FUNCTION ASSEMBLE_LWORD_FROM_DWORDS (* this Function combines the 2 DWORDS to a LWORD *)
  (* Standard: 61499-1; Description: Copyright (c) 2026 HR Agrartechnik GmbH This program and the accompanying materials are made available under the terms of the Eclipse Public License 2.0 which is available at https://www.eclipse.org/legal/epl-2.0/ SPDX-License-Identifier: EPL-2.0 *)
  (* Version 1.0, 2026-05-16, Franz Höpfinger, HR Agrartechnik, initial Implementation *)
  PACKAGE eclipse4diac::utils::assembling;
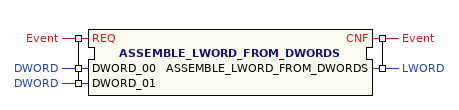
  EVENT_INPUT
    REQ WITH DWORD_00, DWORD_01;
  END_EVENT
  EVENT_OUTPUT
    CNF WITH ASSEMBLE_LWORD_FROM_DWORDS;
  END_EVENT
  VAR_INPUT
    DWORD_00 : DWORD;
    DWORD_01 : DWORD;
  END_VAR
  VAR_OUTPUT
    ASSEMBLE_LWORD_FROM_DWORDS : LWORD;
  END_VAR
  BODY IN ST:
(* this Function combines the 2 DWORDS to a LWORD *)
FUNCTION ASSEMBLE_LWORD_FROM_DWORDS : LWORD

VAR_INPUT
	DWORD_00 : DWORD;
	DWORD_01 : DWORD;
END_VAR

ASSEMBLE_LWORD_FROM_DWORDS.%D0 := DWORD_00;
ASSEMBLE_LWORD_FROM_DWORDS.%D1 := DWORD_01;

END_FUNCTION
  END_BODY
END_FUNCTION
